TYPE ST_PU_Schuetz_Steuerung :
STRUCT
	Freigabe			: ST_Steuerung_auto_manu_BOOL;
	Freigabe_Deakt	: ST_Steuerung_auto_manu_BOOL;
	Betrieb_Anford	: ST_Steuerung_auto_manu_opti_BOOL;
	Quittierung		: BOOL;
END_STRUCT
END_TYPE

(* stored: Version 1.1.0.1, ProductVersion 3.1.4024.9
   DUT ST_PU_Schuetz_Steuerung: Id {073a63dd-c3ff-490c-a4d8-49bddd9d8966} *)
